TYPE ST_HTTP_File_Download_Status :
STRUCT
	Done : BOOL;
	Busy : BOOL;
	Error : BOOL;
	ErrorType : E_HTTP_File_Download_Error;
	Progress : LREAL;
	BytesOfData : ULINT;
	FileSupported : BOOL;
END_STRUCT
END_TYPE

(* stored: Version 1.1.0.1, ProductVersion 3.1.4024.12
   DUT ST_HTTP_File_Download_Status: Id {bdcc0845-344b-4698-a479-cf1753d68e3b} *)
